# EPICS autosave request: iocBoot/ioc14ida/HeatLoadShutter.req
$(P)$(Q)0.DO2
$(P)$(Q)1.DO2
$(P)$(Q)2.DO2
$(P)$(Q)3.DO2
$(P)$(Q)4.DO2
$(P)$(Q)5.DO2
$(P)$(Q)6.DO2
$(P)$(Q)7.DO2
$(P)$(Q)8.DO2
$(P)$(Q)9.DO2
$(P)$(Q)0.DO3
$(P)$(Q)1.DO3
$(P)$(Q)2.DO3
$(P)$(Q)3.DO3
$(P)$(Q)4.DO3
$(P)$(Q)5.DO3
$(P)$(Q)6.DO3
$(P)$(Q)7.DO3
$(P)$(Q)8.DO3
$(P)$(Q)9.DO3
